FUNCTION F_Concat5 : STRING(255)
VAR_INPUT
	sString1: STRING(255);
	sString2: STRING(255);
	sString3: STRING(255);
	sString4: STRING(255);
	sString5: STRING(255);
END_VAR

F_Concat5 := CONCAT(F_Concat5, sString1);
F_Concat5 := CONCAT(F_Concat5, sString2);
F_Concat5 := CONCAT(F_Concat5, sString3);
F_Concat5 := CONCAT(F_Concat5, sString4);
F_Concat5 := CONCAT(F_Concat5, sString5);

END_FUNCTION

(* stored: Version 1.1.0.1, ProductVersion 3.1.4022.18
   POU F_Concat5: Id {fc25d7ea-2259-44d7-8476-49bf315e07e0}, SpecialFunc None *)
